PROGRAM MAIN
VAR
	CMMT_AS_EtherCAT	: CMMT_AS_EtherCAT;
	
END_VAR

CMMT_AS_EtherCAT();

END_PROGRAM

(* stored: Version 1.1.0.1, ProductVersion 3.1.4024.12
   POU MAIN: Id {56d30d04-7a42-4f26-a728-92588274e883}, SpecialFunc None *)
